Omron Sysmac Studio project IkıncıKurs_Basladi (Sysmac Studio 1.65.0.64007, StandardProject)

# Controller new_Controller_0: NX1P2-1040DT1 version 1.69
Task PrimaryTask (priority 4, period or condition 2000): Program0

TYPE Motor : STRUCT
    Start : BOOL;
    Fault : BOOL;
    Ref : REAL;
END_STRUCT END_TYPE
TYPE SYSTEM : STRUCT
    AlwaysTrue : BOOL;
    AlwaysFalse : BOOL;
    FirstCycle : BOOL;
    Pulse_Single_100ms : BOOL;
    Pulse_Single_200ms : BOOL;
    Pulse_Single_300ms : BOOL;
    Pulse_OnOff_100ms : BOOL;
    Pulse_OnOff_200ms : BOOL;
    Pulse_OnOff_300ms : BOOL;
    Year : UINT;
    Month : USINT;
    Day : USINT;
    Hour : USINT;
    Minute : USINT;
    Second : USINT;
END_STRUCT END_TYPE
TYPE uWORD : UNION
    Bits : ARRAY[0..15] OF BOOL;
    Bytes : ARRAY[0..1] OF BYTE;
    Words : WORD;
END_UNION END_TYPE
TYPE uDWORD : UNION
    Bits : ARRAY[0..31] OF BOOL;
    Bytes : ARRAY[0..3] OF BYTE;
    Words : ARRAY[0..1] OF WORD;
    Dwords : DWORD;
END_UNION END_TYPE
TYPE eUsers : (Opr := 0, prg := 1, admin := 2); END_TYPE
TYPE MakineDurum : (Ready := 0, Fault := 1, AutoRunning := 2, ManRunning := 3, Home := 4); END_TYPE

VAR_GLOBAL RETAIN
    SYS : SYSTEM;
    E_DWORD_Value : DWORD;  (* published *)
    E_Invert_DWORD : DWORD;  (* published *)
END_VAR
VAR_GLOBAL
    E_Sifre : DINT;  (* published *)
END_VAR
VAR_GLOBAL RETAIN
    User_Level : DINT;  (* published *)
    MakineDurumm : DINT;  (* published *)
END_VAR

PROGRAM Program0
VAR
    Motor1 : Motor;
    Alarm : BOOL;
    IN_START : BOOL;
    System_Variables : SystemTags;
    E_Actual_Year : UINT;
    IntValue : INT;
    Union_Value : uWORD;
    uVariable1 : uDWORD;
    uVariable2 : uDWORD;
    Tentative_Value_0 : WORD;
    Tentative_Value_1 : WORD;
    eUser_Level : eUsers;
    Makine_Durum : MakineDurum;
    ReadySartlari : BOOL;
    FaultSartlari : BOOL;
    AutoRunningSartlari : BOOL;
    ManRunningSartlari : BOOL;
    HomeSartlari : BOOL;
END_VAR
VAR_EXTERNAL
    SYS : SYSTEM;
    E_DWORD_Value : DWORD;
    E_Invert_DWORD : DWORD;
    E_Sifre : DINT;
    User_Level : DINT;
    MakineDurumm : DINT;
END_VAR

(* Section Main: ladder, written here as Structured Text *)

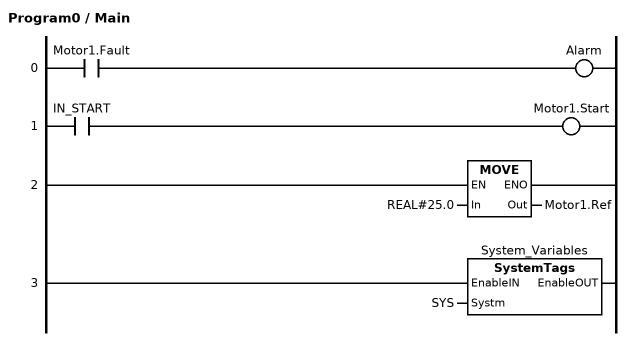
(* Rung 0 *)
Alarm := Motor1.Fault;
(* Rung 1 *)
Motor1.Start := IN_START;
(* Rung 2 *)
Motor1.Ref := REAL#25.0;
(* Rung 3 *)
System_Variables(EnableIN := TRUE, Systm := SYS);

(* Section Section1: ladder, written here as Structured Text *)

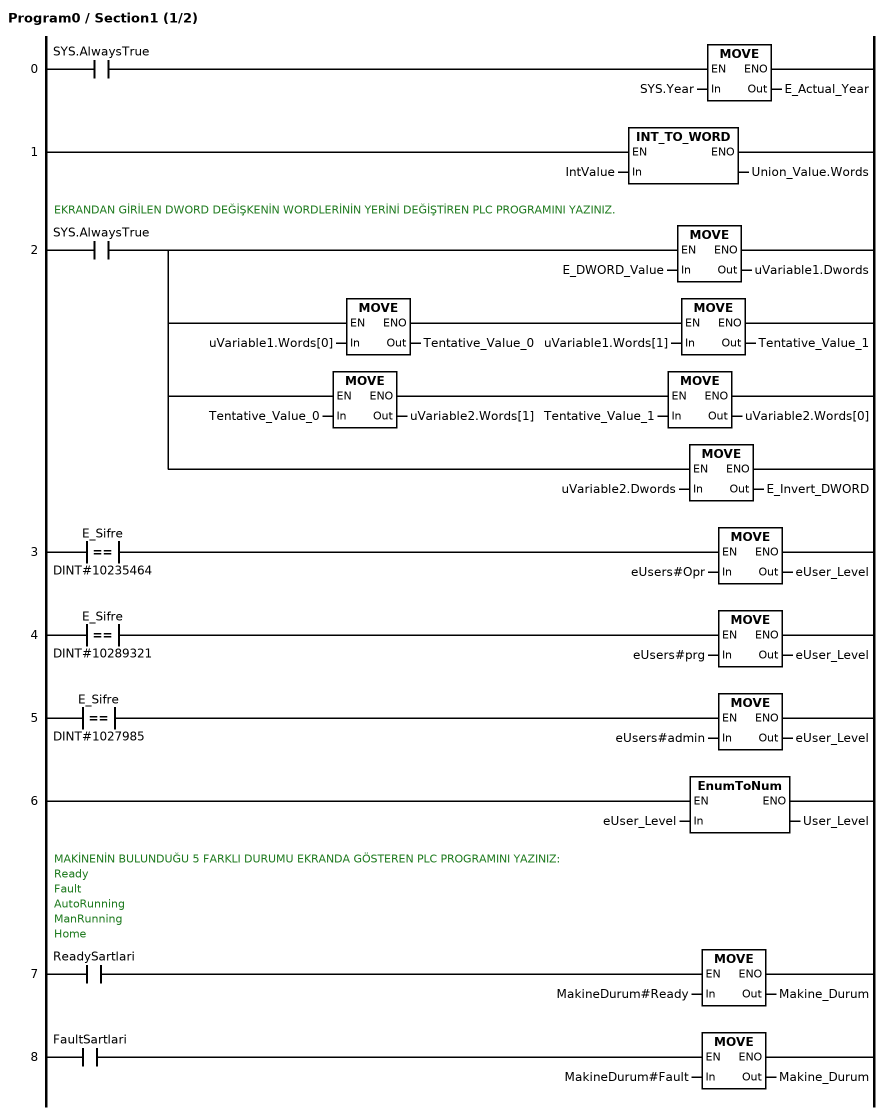
(* Rung 0 *)
IF SYS.AlwaysTrue THEN E_Actual_Year := SYS.Year; END_IF;
(* Rung 1 *)
Union_Value.Words := INT_TO_WORD(In := IntValue);
(* Rung 2: EKRANDAN GİRİLEN DWORD DEĞİŞKENİN WORDLERİNİN YERİNİ DEĞİŞTİREN PLC PROGRAMINI YAZINIZ. *)
IF SYS.AlwaysTrue THEN
    uVariable1.Dwords := E_DWORD_Value;
    Tentative_Value_0 := uVariable1.Words[0];
    Tentative_Value_1 := uVariable1.Words[1];
    uVariable2.Words[1] := Tentative_Value_0;
    uVariable2.Words[0] := Tentative_Value_1;
    E_Invert_DWORD := uVariable2.Dwords;
END_IF;
(* Rung 3 *)
IF E_Sifre = DINT#10235464 THEN eUser_Level := eUsers#Opr; END_IF;
(* Rung 4 *)
IF E_Sifre = DINT#10289321 THEN eUser_Level := eUsers#prg; END_IF;
(* Rung 5 *)
IF E_Sifre = DINT#1027985 THEN eUser_Level := eUsers#admin; END_IF;
(* Rung 6 *)
User_Level := EnumToNum(In := eUser_Level);
(* Rung 7: MAKİNENİN BULUNDUĞU 5 FARKLI DURUMU EKRANDA GÖSTEREN PLC PROGRAMINI YAZINIZ: / Ready / Fault / AutoRunning / ManRunning / Home *)
IF ReadySartlari THEN Makine_Durum := MakineDurum#Ready; END_IF;
(* Rung 8 *)
IF FaultSartlari THEN Makine_Durum := MakineDurum#Fault; END_IF;

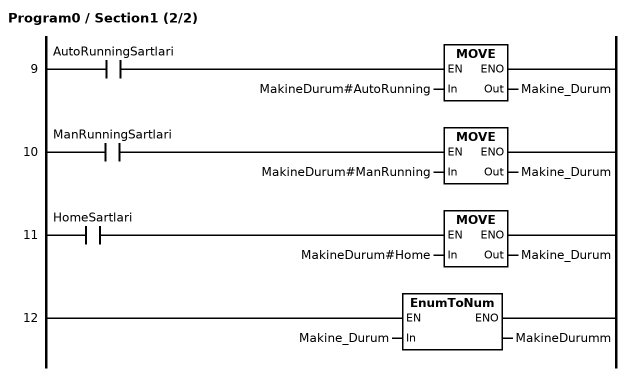
(* Rung 9 *)
IF AutoRunningSartlari THEN Makine_Durum := MakineDurum#AutoRunning; END_IF;
(* Rung 10 *)
IF ManRunningSartlari THEN Makine_Durum := MakineDurum#ManRunning; END_IF;
(* Rung 11 *)
IF HomeSartlari THEN Makine_Durum := MakineDurum#Home; END_IF;
(* Rung 12 *)
MakineDurumm := EnumToNum(In := Makine_Durum);
END_PROGRAM

FUNCTION_BLOCK SystemTags
VAR
    TON_100ms : TON;
    TON_200ms : TON;
    TON_300ms : TON;
    TON_400ms : TON;
    TON_600ms : TON;
    Call_Time : DATE_AND_TIME;
    Date_Struct : _sDT;
END_VAR
VAR_INPUT
    EnableIN : BOOL;
END_VAR
VAR_OUTPUT
    EnableOUT : BOOL;
END_VAR
VAR_IN_OUT
    Systm : SYSTEM;
END_VAR
VAR
    _p1 : BOOL;
    _p2 : BOOL;
    _p3 : BOOL;
    _p4 : BOOL;
    _p5 : BOOL;
END_VAR
(* ladder, written here as Structured Text *)

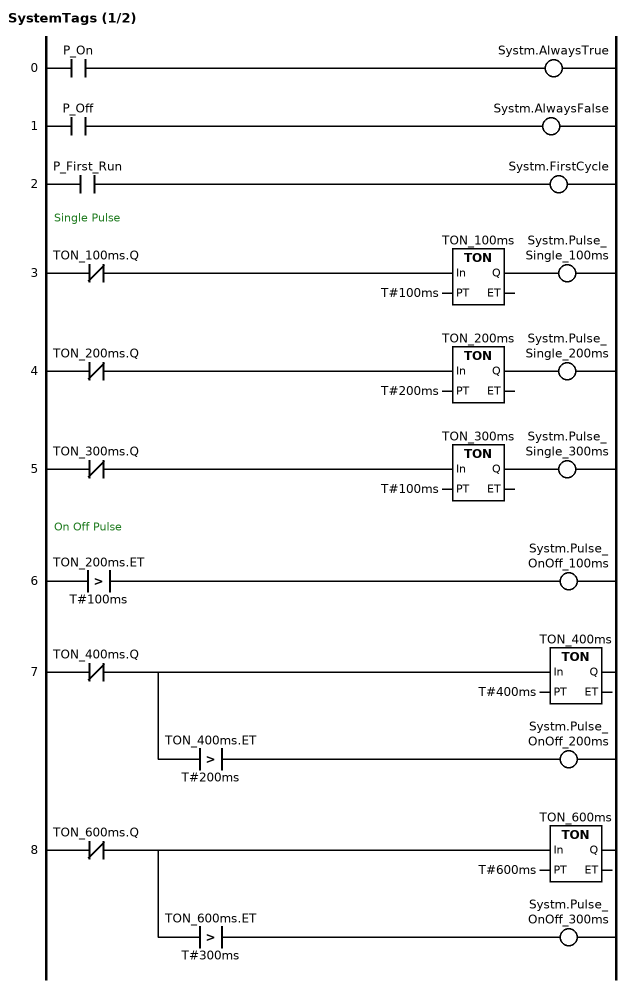
(* Rung 0 *)
Systm.AlwaysTrue := P_On;
(* Rung 1 *)
Systm.AlwaysFalse := P_Off;
(* Rung 2 *)
Systm.FirstCycle := P_First_Run;
(* Rung 3: Single Pulse *)
_p1 := NOT TON_100ms.Q;
TON_100ms(In := _p1, PT := T#100ms);
Systm.Pulse_Single_100ms := TON_100ms.Q;
(* Rung 4 *)
_p2 := NOT TON_200ms.Q;
TON_200ms(In := _p2, PT := T#200ms);
Systm.Pulse_Single_200ms := TON_200ms.Q;
(* Rung 5 *)
_p3 := NOT TON_300ms.Q;
TON_300ms(In := _p3, PT := T#100ms);
Systm.Pulse_Single_300ms := TON_300ms.Q;
(* Rung 6: On Off Pulse *)
Systm.Pulse_OnOff_100ms := TON_200ms.ET > T#100ms;
(* Rung 7 *)
_p4 := NOT TON_400ms.Q;
TON_400ms(In := _p4, PT := T#400ms);
Systm.Pulse_OnOff_200ms := _p4 AND (TON_400ms.ET > T#200ms);
(* Rung 8 *)
_p5 := NOT TON_600ms.Q;
TON_600ms(In := _p5, PT := T#600ms);
Systm.Pulse_OnOff_300ms := _p5 AND (TON_600ms.ET > T#300ms);

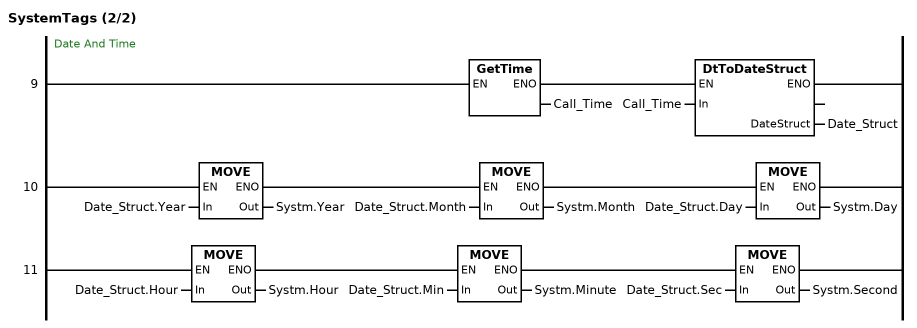
(* Rung 9: Date And Time *)
Call_Time := GetTime();
DtToDateStruct(In := Call_Time, DateStruct => Date_Struct);
(* Rung 10 *)
Systm.Year := Date_Struct.Year;
Systm.Month := Date_Struct.Month;
Systm.Day := Date_Struct.Day;
(* Rung 11 *)
Systm.Hour := Date_Struct.Hour;
Systm.Minute := Date_Struct.Min;
Systm.Second := Date_Struct.Sec;
END_FUNCTION_BLOCK